TYPE ServicesConfig :
STRUCT
	///Timing config
	timing: ServicesTimingConfig;
END_STRUCT
END_TYPE

(* stored: Version 1.1.0.1, ProductVersion 3.1.4019.2
   DUT ServicesConfig: Id {63e3cc66-92f2-4f94-97d8-088350a457ba} *)
